FUNCTION_BLOCK Section4
  (* Standard: 61499-2 *)
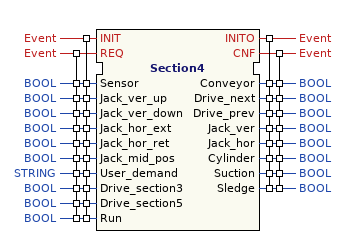
  EVENT_INPUT
    INIT WITH Sensor, Jack_ver_up, Jack_ver_down, Jack_hor_ext, Jack_hor_ret, Jack_mid_pos, User_demand, Drive_section3, Drive_section5, Run;
    REQ WITH Sensor, Jack_ver_up, Jack_ver_down, Jack_hor_ext, Jack_hor_ret, Jack_mid_pos, User_demand, Drive_section3, Drive_section5, Run;
  END_EVENT
  EVENT_OUTPUT
    INITO WITH Conveyor, Drive_next, Drive_prev, Jack_ver, Jack_hor, Cylinder, Suction, Sledge;
    CNF WITH Conveyor, Drive_next, Drive_prev, Jack_ver, Jack_hor, Cylinder, Suction, Sledge;
  END_EVENT
  VAR_INPUT
    Sensor : BOOL;
    Jack_ver_up : BOOL;
    Jack_ver_down : BOOL;
    Jack_hor_ext : BOOL;
    Jack_hor_ret : BOOL;
    Jack_mid_pos : BOOL;
    User_demand : STRING;
    Drive_section3 : BOOL;
    Drive_section5 : BOOL;
    Run : BOOL;
  END_VAR
  VAR_OUTPUT
    Conveyor : BOOL;
    Drive_next : BOOL;
    Drive_prev : BOOL;
    Jack_ver : BOOL;
    Jack_hor : BOOL;
    Cylinder : BOOL;
    Suction : BOOL;
    Sledge : BOOL;
  END_VAR
  FBS
    FB2 : DisableConveyor;
    Section4Ctrl : Section4Ctrl;
    Jack2Ctrl : Jack2Ctrl;
  END_FBS
  EVENT_CONNECTIONS
    INIT TO Section4Ctrl.INIT;
    REQ TO Section4Ctrl.REQ;
    Section4Ctrl.INITO TO FB2.INIT;
    Section4Ctrl.CNF TO FB2.REQ;
    Section4Ctrl.CNF TO Jack2Ctrl.REQ;
    INIT TO Jack2Ctrl.INIT;
    Jack2Ctrl.CNF TO Section4Ctrl.REQ;
    REQ TO FB2.REQ;
    FB2.CNF TO CNF;
    REQ TO Jack2Ctrl.REQ;
  END_CONNECTIONS
  DATA_CONNECTIONS
    Sensor TO Section4Ctrl.Sensor;
    Jack_ver_up TO Jack2Ctrl.JackVerUp;
    Jack_ver_down TO Jack2Ctrl.JackVerDown;
    Jack_hor_ext TO Jack2Ctrl.JackHorExt;
    Jack_hor_ret TO Jack2Ctrl.JackHorRet;
    Jack_mid_pos TO Jack2Ctrl.JackMidPos;
    User_demand TO Jack2Ctrl.User_demand;
    Section4Ctrl.Conveyor TO FB2.ConvIn;
    Section4Ctrl.Jack2_produces TO Jack2Ctrl.Produce_SIG;
    Jack2Ctrl.ReadySIG TO Section4Ctrl.Jack2_finished;
    Run TO FB2.QI;
    Drive_section3 TO Section4Ctrl.Drive_section3;
    Drive_section5 TO Section4Ctrl.Drive_section5;
    Jack2Ctrl.JackVer TO Jack_ver;
    Jack2Ctrl.JackHor TO Jack_hor;
    Jack2Ctrl.Cylinder TO Cylinder;
    Jack2Ctrl.Suction TO Suction;
    Jack2Ctrl.Sledge TO Sledge;
    FB2.ConvOut TO Conveyor;
    Section4Ctrl.Drive_next TO Drive_next;
    Section4Ctrl.Drive_prev TO Drive_prev;
  END_CONNECTIONS
END_FUNCTION_BLOCK
